DATA_BLOCK "DB1_C"
{ S7_Optimized_Access := 'TRUE' }
NAME : FCDI
VERSION : 0.1
NON_RETAIN
"FB1_C"

BEGIN
   dnCALLCHECK_C := 61159;
   dnTRACER_START := 20389;
   dnGCTX_DBNUMBER := 30010;

END_DATA_BLOCK

